(* PLC project Sin nombre, Desconocido Sin nombre 1 *)
(* stored: creationDateTime 2025-10-23T16:17:31, modificationDateTime 2025-10-23T18:00:32 *)

PROGRAM main
  VAR
    Inclinacion AT I0.7 : BOOL := FALSE;  (* Sensor de inclinacion *)
    LedVerde AT Q0.6 : BOOL := TRUE;  (* Led verde *)
    LedRojo AT Q0.5 : BOOL := FALSE;  (* Led rojo *)
    Rele AT Q0.4 : BOOL := FALSE;  (* Rele *)
  END_VAR

(* LD diagram, written out as Structured Text *)
Inclinacion := Inclinacion;
Inclinacion := NOT Inclinacion;
(* drawn but not wired to any output: LedVerde, LedRojo, Rele *)
END_PROGRAM

CONFIGURATION Config0
  RESOURCE Res0 ON PLC
    TASK task0(INTERVAL := T#20ms, PRIORITY := 0);
    PROGRAM instance0 WITH task0 : main;
  END_RESOURCE
END_CONFIGURATION
